// TIA Portal V20 export
// export: Created 2026-04-18T06:33:56.6715178Z, ExportSetting WithDefaults, DisplayName Totally Integrated Automation Portal, DisplayVersion V20, DisplayName TIA Portal Openness, DisplayVersion V20, DisplayName TIA Portal Version Control Interface, DisplayVersion V20, DisplayName STEP 7 Professional, DisplayVersion V20, DisplayName STEP 7 Safety, DisplayVersion V20, DisplayName WinCC Basic/Comfort/Advanced, DisplayVersion V20
TYPE "UDT_EquipmentModule"
// stored: IsFailsafeCompliant false
   STRUCT
      moduleId : Int := 0;
      moduleName : String[32] := 'Module';
      moduleType : Int := 1;   // 1=Dosing 2=Heating 3=Stirring 4=Draining
      valves { S7_SetPoint := 'True'} : Array[1..4] of "UDT_ControlValve";
   END_STRUCT;
END_TYPE
